// TIA Portal project "Verbinder_Station_0" (V20)

(* hardware
DEVICE "S7-1500/ET200MP-Station_1"  S7-1500 station
   slot 0: "Profilschiene_0"  Rack  6ES7 590-1***0-0AA0
   slot 1: "PLC_1"  CPU 1513-1 PN  6ES7 513-1AM03-0AB0  V4.0
      slot 3: "CPU-Display_1"  6ES7591-1AA00-0AA0
      slot 32768: "PROFINET-Schnittstelle_1"  X1
         slot 32769: "Port_1"  X1 P1
         slot 32770: "Port_2"  X1 P2
      slot 34817: "Virtual CP interface port_1"  Virtual CP interface port  Virtual CP interface port FW V4.0
   slot 2: "DI 16x24VDC BA_1"  DI 16x24VDC BA  6ES7 521-1BH10-0AA0  V1.1
   slot 3: "DQ 16x24VDC/0.5A ST_1"  DQ 16x24VDC/0.5A ST  6ES7 522-1BH00-0AB0  V2.0
   slot 4: "AI 8xU/I/R/RTD BA_1"  AI 8xU/I/R/RTD BA  6ES7 531-7QF00-0AB0  V1.0
   slot 5: "AQ 8xU/I HS_1"  AQ 8xU/I HS  6ES7 532-5HF00-0AB0  V2.2
   slot 6: "AQ 8xU/I HS_2"  AQ 8xU/I HS  6ES7 532-5HF00-0AB0  V2.2
*)

// ===== PLC "PLC_1"  CPU 1513-1 PN =====

VAR_GLOBAL   // PLC tag table "Standard-Variablentabelle"
   "PlcLabConnectIn01" AT %ID32760 : DWord;
   "PlcLabConnectIn02" AT %ID32764 : DWord;
   "PlcLabConnectOut01" AT %QD32760 : DWord;
   "PlcLabConnectOut02" AT %QD32764 : DWord;
   "NotAus_aktiv" AT %M1.0 : Bool;
   "Bänder_laufen" AT %M1.1 : Bool;
   "Clock_Byte" AT %MB0 : Byte;
   "Clock_10Hz" AT %M0.0 : Bool;
   "Clock_5Hz" AT %M0.1 : Bool;
   "Clock_2.5Hz" AT %M0.2 : Bool;
   "Clock_2Hz" AT %M0.3 : Bool;
   "Clock_1.25Hz" AT %M0.4 : Bool;
   "Clock_1Hz" AT %M0.5 : Bool;
   "Clock_0.625Hz" AT %M0.6 : Bool;
   "Clock_0.5Hz" AT %M0.7 : Bool;
   "Einlauf_1_aktiv" AT %M2.0 : Bool;
   "Einlauf_2_aktiv" AT %M2.1 : Bool;
   "Transfer_2_zu_1" AT %M2.2 : Bool;
   "Palette_vorbei" AT %M2.7 : Bool;
   "Transfer_1_belegt" AT %M1.2 : Bool;
   "Transfer_2_frei" AT %M1.3 : Bool;
   "Transfer_starten" AT %M1.4 : Bool;
   "1b1_Palette" AT %M2.3 : Bool;
   "2b1_Palette" AT %M2.4 : Bool;
   "3b1_Palette" AT %M2.5 : Bool;
   "Tag_1" AT %M1.6 : Bool;
   "Tag_2" AT %M1.7 : Bool;
END_VAR

VAR_GLOBAL   // PLC tag table "Eingaenge"
   "S1" AT %E0.0 : Bool;   // Not-Aus
   "S2" AT %E0.1 : Bool;   // Betriebsschalter
   "S3" AT %I0.2 : Bool;   // Starttaster
   "S4" AT %I0.3 : Bool;   // Stoptaster
   "S5" AT %I0.4 : Bool;   // Reset
   "1B1" AT %I1.0 : Bool;   // Sensor Ein 1
   "1B2" AT %I1.1 : Bool;   // Endanschlag 1
   "2B1" AT %I1.2 : Bool;   // Sensor Ein 2
   "2B2" AT %I1.3 : Bool;   // Endanschlag 2
   "3B1" AT %I1.4 : Bool;   // Sensor Aus
END_VAR

VAR_GLOBAL   // PLC tag table "Ausgaenge"
   "H1" AT %Q0.2 : Bool;   // Start Leuchte
   "H2" AT %Q0.3 : Bool;   // Stop Leuchte
   "H3" AT %Q0.4 : Bool;   // Reset Leuchte
   "M1" AT %Q1.0 : Bool;   // Band Ein 1
   "M2" AT %Q1.1 : Bool;   // Band Ein 2
   "M3" AT %Q1.2 : Bool;   // Laden 1
   "M4" AT %Q1.3 : Bool;   // Laden 2
   "M5" AT %Q1.4 : Bool;   // Band Aus
   "M6" AT %Q1.5 : Bool;   // Transfer 1
   "M7" AT %Q1.6 : Bool;   // Transfer 2
   "D1" AT %QD30 : DInt;   // Zähler
END_VAR

// folder: System blocks/Program resources

DATA_BLOCK "IEC_Counter_0_DB"   // DB1
{ S7_Optimized_Access := 'TRUE' }
AUTHOR : SIMATIC
FAMILY : IEC
NAME : DCNTR
VERSION : 1.2
// stored: InstanceOfName IEC_DCOUNTER
"IEC_DCOUNTER"
BEGIN
END_DATA_BLOCK

// folder: (top level)

FUNCTION "Rollensteuerung" : Void   // FC1, FBD
{ S7_Optimized_Access := 'TRUE' }
VERSION : 0.1
   VAR_TEMP   // added for the SCL form of the ladder/FBD networks
      _w1 : Bool;
      _w2 : Bool;
      _w3 : Bool;
   END_VAR
BEGIN

REGION Network 1: Bandsteuerung
   // Wenn der Betriebsschalter ein ist und der Not-Aus und Stop nicht aktiv. Dann soll das Auslauf-Förderband immer laufen. Die beiden Einlauf-Förderbänder sollen dann nur aktiv sein, wenn beide Transfer-Stationen frei sind. Und gerade kein Transfer statt findet.
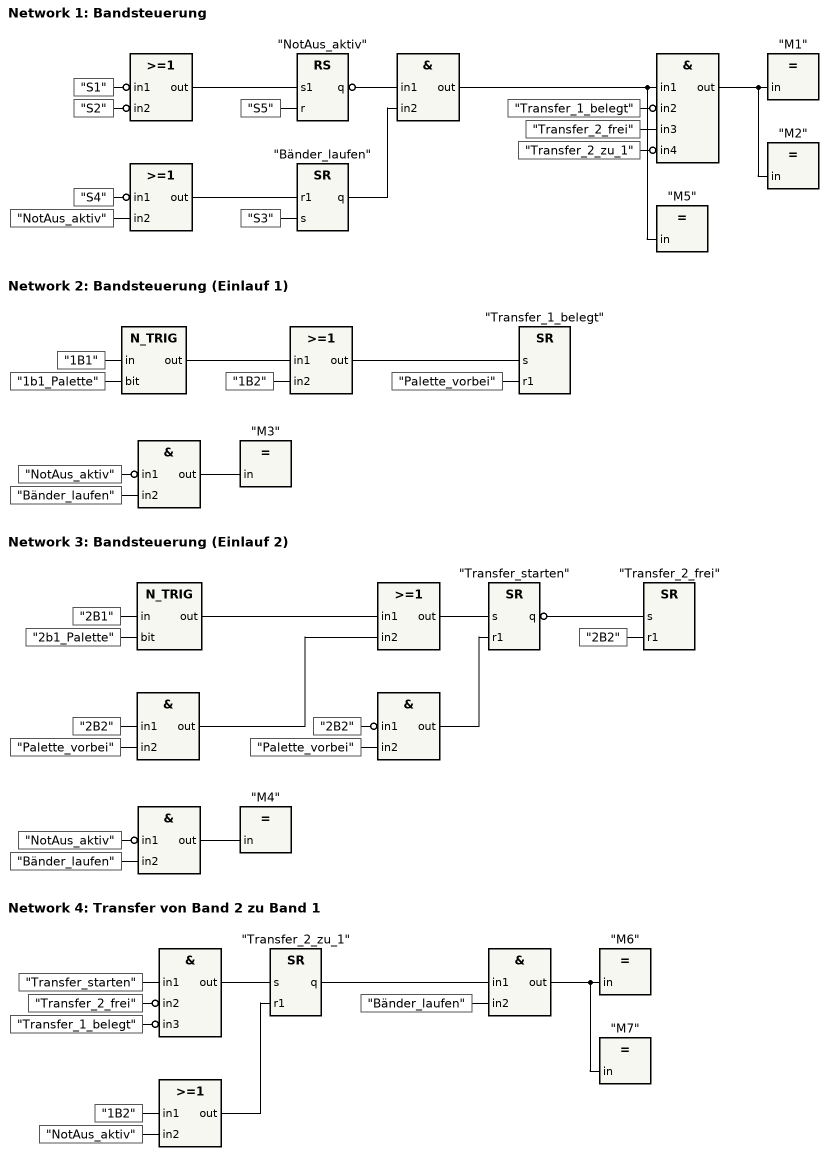
   IF "S5" THEN
       "NotAus_aktiv" := FALSE;   // RS flip-flop
   END_IF;
   IF NOT "S1" OR NOT "S2" THEN "NotAus_aktiv" := TRUE; END_IF;
   IF "S3" THEN
       "Bänder_laufen" := TRUE;   // SR flip-flop
   END_IF;
   IF NOT "S4" OR "NotAus_aktiv" THEN "Bänder_laufen" := FALSE; END_IF;
   #_w1 := NOT "NotAus_aktiv" AND "Bänder_laufen";
   "M1" := #_w1 AND NOT "Transfer_1_belegt" AND "Transfer_2_frei" AND NOT "Transfer_2_zu_1";
   "M2" := "M1";
   "M5" := #_w1;
END_REGION

REGION Network 2: Bandsteuerung (Einlauf 1)
   // Solange die Anlage an ist, soll die Transferstation neue Paletten aufnehmen. Sobald eine Palette in der Station ist (vom Einlaufband oder durch Transfer), setze den Merker, dass diese belegt ist. Wenn die Palette aus der Station raus ist, setzte diesen zurück.
   #_w1 := NOT "1B1" AND "1b1_Palette";   // falling edge
   "1b1_Palette" := "1B1";
   IF #_w1 OR "1B2" THEN
       "Transfer_1_belegt" := TRUE;   // SR flip-flop
   END_IF;
   IF "Palette_vorbei" THEN "Transfer_1_belegt" := FALSE; END_IF;
   "M3" := NOT "NotAus_aktiv" AND "Bänder_laufen";
END_REGION

REGION Network 3: Bandsteuerung (Einlauf 2)
   // Solange die Anlage an ist, soll die Transferstation neue Paletten aufnehmen. Sobald eine Palette in der Station ist (vom Einlaufband) und die andere Transferstation frei ist, setze den Merker, dass der Transfer starten soll und dass die Station belegt ist. Wenn die Palette aus der Station raus ist, setzte diesen zurück.
   #_w1 := NOT "2B1" AND "2b1_Palette";   // falling edge
   "2b1_Palette" := "2B1";
   IF #_w1 OR ("2B2" AND "Palette_vorbei") THEN
       "Transfer_starten" := TRUE;   // SR flip-flop
   END_IF;
   IF NOT "2B2" AND "Palette_vorbei" THEN "Transfer_starten" := FALSE; END_IF;
   IF NOT "Transfer_starten" THEN
       "Transfer_2_frei" := TRUE;   // SR flip-flop
   END_IF;
   IF "2B2" THEN "Transfer_2_frei" := FALSE; END_IF;
   "M4" := NOT "NotAus_aktiv" AND "Bänder_laufen";
END_REGION

REGION Network 4: Transfer von Band 2 zu Band 1
   // Sobald der Transfer gestartet werden soll und auf Station 1 keine Palette ist und auf Station 2 eine Palette ist, starte den Transfer von Station 2 zu 1. Tue dies nur solange, wie die Palette Station 1 noch nicht erreicht hat und wenn kein Stop oder Not-Aus aktiv ist.
   IF "Transfer_starten" AND NOT "Transfer_2_frei" AND NOT "Transfer_1_belegt" THEN
       "Transfer_2_zu_1" := TRUE;   // SR flip-flop
   END_IF;
   IF "1B2" OR "NotAus_aktiv" THEN "Transfer_2_zu_1" := FALSE; END_IF;
   "M6" := "Transfer_2_zu_1" AND "Bänder_laufen";
   "M7" := "M6";
END_REGION

REGION Network 5: Palettenzähler
   // Zähle hoch, wenn eine Palette den Auslaufsensor passiert hat. Der Zähler wird über den Resettaster zurückgesetzt. Sobald eine neue Palette die Station erreicht, setzte den Merker zurück, dass gerade keine Palette in der Station ist.
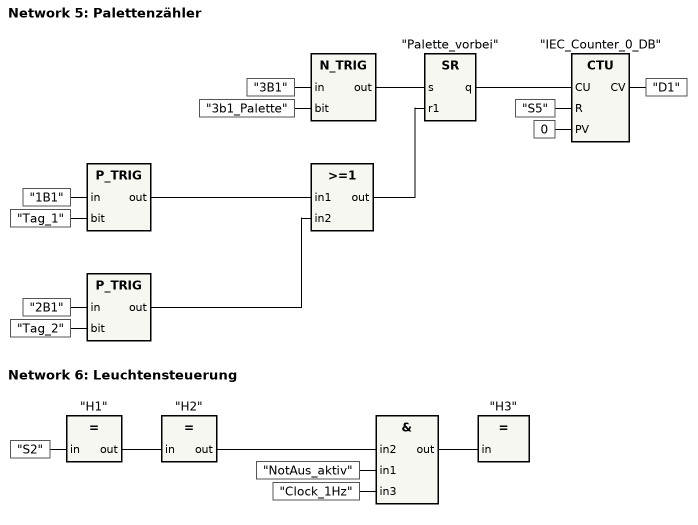
   #_w1 := NOT "3B1" AND "3b1_Palette";   // falling edge
   "3b1_Palette" := "3B1";
   #_w2 := "1B1" AND NOT "Tag_1";   // rising edge
   "Tag_1" := "1B1";
   #_w3 := "2B1" AND NOT "Tag_2";   // rising edge
   "Tag_2" := "2B1";
   IF #_w1 THEN
       "Palette_vorbei" := TRUE;   // SR flip-flop
   END_IF;
   IF #_w2 OR #_w3 THEN "Palette_vorbei" := FALSE; END_IF;
   "IEC_Counter_0_DB".CTU(CU := "Palette_vorbei", R := "S5", PV := 0, CV => "D1");
END_REGION

REGION Network 6: Leuchtensteuerung
   // Die Reset Taste soll blinken, wenn die Anlage an ist und der Not-Aus aktiv ist. Die anderen Leuchten sollen an sein, wenn die Anlage an ist.
   "H1" := "S2";
   "H2" := "S2";
   "H3" := "S2" AND "NotAus_aktiv" AND "Clock_1Hz";
END_REGION
END_FUNCTION

ORGANIZATION_BLOCK "Main"   // OB1, FBD, ProgramCycle
TITLE = "Main Program Sweep (Cycle)"
{ S7_Optimized_Access := 'TRUE' }
VERSION : 0.1
   VAR_INPUT
      Initial_Call : Bool;   // Initial call of this OB
      Remanence : Bool;   // =True, if remanent data are available
   END_VAR
BEGIN

REGION Network 1
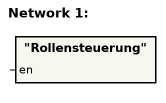
   "Rollensteuerung"();
END_REGION
END_ORGANIZATION_BLOCK